(* IEC 61131-3 sources: controlforge-structured-text/manual-tests/diagnostics, 6 files *)

(* ---- array-bounds.st ---- *)
(* Manual QA: array bounds checking for constant indices *)
(* Open this file in VS Code. Verify red squiggles appear ONLY on lines marked  *)
(* "EXPECT ERROR" and that no errors appear on lines marked "OK".               *)
(* Check the Problems panel (Ctrl+Shift+M) for full messages.                   *)

PROGRAM ArrayBoundsTest
VAR
    temps    : ARRAY[1..10] OF REAL;     (* bounds: 1 to 10 *)
    buf      : ARRAY[0..7]  OF BYTE;     (* bounds: 0 to 7  *)
    offsets  : ARRAY[-5..5] OF INT;      (* bounds: -5 to 5 *)
    matrix   : ARRAY[1..4, 1..4] OF REAL; (* 2-D: rows 1-4, cols 1-4 *)
    i        : INT;
    x        : REAL;
END_VAR

    (* --- single-dimension, 1-based --- *)

    (* OK: boundary values *)
    temps[1]  := 20.0;
    temps[10] := 99.9;
    temps[5]  := 50.0;

    (* EXPECT ERROR: index 0 below lower bound 1
       Message: Array index 0 is out of bounds [1..10] for 'temps' *)
    temps[0] := 10.0;

    (* EXPECT ERROR: index 11 above upper bound 10
       Message: Array index 11 is out of bounds [1..10] for 'temps' *)
    temps[11] := 10.0;

    (* EXPECT ERROR: index 15 far above upper bound
       Message: Array index 15 is out of bounds [1..10] for 'temps' *)
    temps[15] := 25.0;

    (* OK: variable index — not checked *)
    temps[i] := 0.0;

    (* --- zero-based array --- *)

    (* OK: valid range *)
    buf[0] := 0;
    buf[7] := 255;

    (* EXPECT ERROR: index 8 above upper bound 7
       Message: Array index 8 is out of bounds [0..7] for 'buf' *)
    buf[8] := 128;

    (* --- negative lower bound --- *)

    (* OK: valid range *)
    offsets[-5] := -1;
    offsets[0]  :=  0;
    offsets[5]  :=  1;

    (* EXPECT ERROR: index -6 below lower bound -5
       Message: Array index -6 is out of bounds [-5..5] for 'offsets' *)
    offsets[-6] := 0;

    (* EXPECT ERROR: index 6 above upper bound 5
       Message: Array index 6 is out of bounds [-5..5] for 'offsets' *)
    offsets[6] := 0;

    (* --- multi-dimensional array --- *)

    (* OK: all indices in range *)
    matrix[1, 1] := 0.0;
    matrix[4, 4] := 1.0;
    matrix[2, 3] := 0.5;

    (* EXPECT ERROR: first index 0 out of [1..4]
       Message: Array index 0 is out of bounds [1..4] for 'matrix' *)
    matrix[0, 2] := 1.0;

    (* EXPECT ERROR: second index 5 out of [1..4]
       Message: Array index 5 is out of bounds [1..4] for 'matrix' *)
    matrix[2, 5] := 1.0;

    (* --- reading (RHS) also checked --- *)

    (* OK *)
    x := temps[3];

    (* EXPECT ERROR: index 99 out of [1..10]
       Message: Array index 99 is out of bounds [1..10] for 'temps' *)
    x := temps[99];

END_PROGRAM

(* ---- assignment-confusion.st ---- *)
(* Manual QA: := vs = confusion detection *)
(* Open this file in VS Code. Verify yellow squiggles (warnings) appear ONLY   *)
(* on lines marked "EXPECT WARNING" and that no warnings appear on "OK" lines. *)
(* For each warning, a lightbulb quick-fix should be available (Ctrl+.).        *)

PROGRAM AssignmentConfusion
VAR
    counter : INT := 0;
    x       : INT := 5;
    ok      : BOOL;
    tmr     : TON;
    arr     : ARRAY[0..9] OF INT;
END_VAR

    (* === Case 1: '=' in statement context — should be ':=' === *)

    (* EXPECT WARNING: "Used '=' in statement context; did you mean ':='?" *)
    (* Quick-fix: Replace '=' with ':='                                    *)
    counter = counter + 1;

    (* EXPECT WARNING *)
    x = 42;

    (* EXPECT WARNING: array element *)
    arr[0] = 5;

    (* OK: correct := assignment — no warning *)
    counter := counter + 1;
    x := 42;
    arr[0] := 5;

    (* OK: '=' in IF condition — intentional comparison *)
    IF x = 10 THEN
        x := 0;
    END_IF;

    (* OK: '=' inside parentheses (RHS comparison) *)
    ok := (x = 5);

    (* OK: '<=' and '>=' — not a bare '=' *)
    ok := x <= 10;
    ok := x >= 0;

    (* OK: '<>' — not a bare '=' *)
    ok := x <> 0;

    (* OK: '=' inside FB call paren (depth > 0) *)
    tmr(IN := TRUE, PT := T#1s);
    IF tmr.Q = TRUE THEN
        tmr(IN := FALSE, PT := T#1s);
    END_IF;

    (* === Case 2: ':=' in boolean condition — should be '=' === *)

    (* EXPECT WARNING: "Used ':=' in condition context; did you mean '='?" *)
    (* Quick-fix: Replace ':=' with '='                                    *)
    IF x := 10 THEN
        x := 0;
    END_IF;

    (* EXPECT WARNING: in ELSIF *)
    IF x = 0 THEN
        x := 1;
    ELSIF x := 5 THEN
        x := 0;
    END_IF;

    (* EXPECT WARNING: in WHILE *)
    WHILE x := 0 DO
        x := x + 1;
    END_WHILE;

    (* OK: correct '=' in IF condition — no warning *)
    IF x = 10 THEN
        x := 0;
    END_IF;

    (* OK: ':=' in FOR loop header is correct syntax — no warning *)
    FOR x := 1 TO 10 DO
        counter := counter + 1;
    END_FOR;

    (* OK: ':=' inside parens in IF body (named parameter) — no warning *)
    IF tmr.Q = TRUE THEN
        tmr(IN := FALSE, PT := T#1s);
    END_IF;

END_PROGRAM

(* ---- code-action-fixes.st ---- *)
(* Test: Code actions for semantic diagnostics *)
(* Open this file, then use Ctrl+. on squiggles to verify quick fixes *)

(* === Insert Semicolon === *)
(* Expected: Quick fix to insert ';' *)
PROGRAM SemicolonFixTest
VAR
    x : INT;
END_VAR
    x := 1  (* <-- hover, Ctrl+. should offer "Insert semicolon" *)
END_PROGRAM

(* === Remove Duplicate Declaration === *)
(* Expected: Quick fix to remove the duplicate line *)
PROGRAM DuplicateFixTest
VAR
    value : INT;
    value : REAL;  (* <-- Ctrl+. should offer "Remove duplicate declaration" *)
END_VAR
    value := 0;
END_PROGRAM

(* === Remove Unused Variable === *)
(* Expected: Quick fix to remove the unused variable line *)
PROGRAM UnusedFixTest
VAR
    active : BOOL;
    unused : INT;  (* <-- Ctrl+. should offer "Remove unused variable" *)
END_VAR
    active := TRUE;
END_PROGRAM

(* ---- constant-assignment.st ---- *)
(* Manual QA: constant assignment detection *)
(* Open this file in VS Code. Verify red squiggles appear ONLY on the lines   *)
(* marked "EXPECT ERROR" and that no errors appear on lines marked "OK".       *)

(* === VAR_GLOBAL CONSTANT === *)
VAR_GLOBAL CONSTANT
    MAX_TEMP : REAL := 100.0;   (* constant — never writable *)
    VERSION  : STRING := 'v1.0';
END_VAR

VAR_GLOBAL
    currentTemp : REAL := 20.0; (* NOT constant — writable *)
END_VAR

(* === PROGRAM body === *)
(* Open this file, then look at the Problems panel (Ctrl+Shift+M).             *)
PROGRAM ConstantTest
VAR CONSTANT
    PI : REAL := 3.14159;       (* local constant *)
END_VAR
VAR
    result : REAL;
    flag   : BOOL;
END_VAR

    (* EXPECT ERROR: Cannot assign to constant 'MAX_TEMP' *)
    MAX_TEMP := 200.0;

    (* EXPECT ERROR: Cannot assign to constant 'PI' *)
    PI := 3.0;

    (* EXPECT ERROR: Cannot assign to constant 'VERSION' *)
    VERSION := 'v2.0';

    (* OK: regular variable assignment — no error *)
    currentTemp := 50.0;
    result := PI * 2.0;         (* reading PI is fine *)
    flag := currentTemp > MAX_TEMP; (* reading constants is fine *)

    (* OK: named FB parameter that happens to use := inside parens — no error *)
    (* (no FB instance here, but illustrates the paren-depth guard)            *)

END_PROGRAM

(* === Verify no false positives for plain VAR_GLOBAL === *)
PROGRAM NoFalsePositives
VAR
    x : REAL;
END_VAR
    (* OK: currentTemp is NOT constant *)
    currentTemp := 99.0;
    x := currentTemp;
END_PROGRAM

(* ---- for-loop-bounds.st ---- *)
(* Manual QA: FOR loop bounds validation *)
(* Open this file in VS Code. Verify squiggles appear ONLY on lines marked     *)
(* "EXPECT <SEVERITY>" and that no squiggles appear on lines marked "OK".      *)
(* Check the Problems panel (Ctrl+Shift+M) for full messages.                   *)

PROGRAM ForLoopBoundsTest
VAR
    i     : INT;
    start : INT;
    stop  : INT;
    total : INT;
END_VAR

    (* ── Normal ascending loops — no diagnostic expected ─────────────────── *)

    (* OK: ascending, default BY (+1) *)
    FOR i := 1 TO 10 DO
        total := total + i;
    END_FOR;

    (* OK: ascending, explicit BY 1 *)
    FOR i := 1 TO 10 BY 1 DO
        total := total + i;
    END_FOR;

    (* OK: descending with BY -1 *)
    FOR i := 10 TO 1 BY -1 DO
        total := total + i;
    END_FOR;

    (* OK: large positive step still valid direction *)
    FOR i := 0 TO 100 BY 5 DO
        total := total + i;
    END_FOR;

    (* OK: variable bounds — not checked at all *)
    FOR i := start TO stop DO
        total := total + i;
    END_FOR;

    (* OK: negative bounds, descending *)
    FOR i := -1 TO -10 BY -1 DO
        total := total + i;
    END_FOR;

    (* ── BY 0: error ─────────────────────────────────────────────────────── *)

    (* EXPECT ERROR on "BY 0": infinite loop
       Problems panel: "FOR loop step BY 0 causes an infinite loop"           *)
    FOR i := 1 TO 10 BY 0 DO
        total := total + i;
    END_FOR;

    (* ── Reverse range with positive BY: warning ─────────────────────────── *)

    (* EXPECT WARNING on "FOR": loop body never executes
       Problems panel: "FOR loop body never executes: counting up (BY 1) but start (10) > end (1)..." *)
    FOR i := 10 TO 1 BY 1 DO
        total := total + i;
    END_FOR;

    (* EXPECT WARNING on "FOR": default BY (+1) with descending range
       Problems panel: "FOR loop body never executes: counting up (BY 1) but start (10) > end (1)..." *)
    FOR i := 10 TO 1 DO
        total := total + i;
    END_FOR;

    (* EXPECT WARNING on "FOR": ascending range with negative step
       Problems panel: "FOR loop body never executes: counting down (BY -2) but start (1) < end (10)..." *)
    FOR i := 1 TO 10 BY -2 DO
        total := total + i;
    END_FOR;

    (* ── Start equals end: hint ──────────────────────────────────────────── *)

    (* EXPECT HINT on "FOR": executes exactly once — likely unintended
       Problems panel: "FOR loop executes exactly once (start equals end: 5)" *)
    FOR i := 5 TO 5 DO
        total := total + i;
    END_FOR;

    (* EXPECT HINT on "FOR": same with explicit BY
       Problems panel: "FOR loop executes exactly once (start equals end: 3)" *)
    FOR i := 3 TO 3 BY 1 DO
        total := total + i;
    END_FOR;

END_PROGRAM

(* ---- semantic-checks.st ---- *)
(* Test: Semantic diagnostics - Phase 2 checks *)
(* Open this file in VS Code to verify diagnostics appear correctly *)

(* === Missing Semicolons === *)
(* Expected: Error on line with missing semicolon *)
PROGRAM MissingSemicolonTest
VAR
    x : INT := 0;
    y : INT := 0;
END_VAR
    x := 1;
    y := x + 2  (* <-- missing semicolon, should show error *)
END_PROGRAM

(* === Duplicate Declarations === *)
(* Expected: Error on second declaration of 'counter' *)
PROGRAM DuplicateVarTest
VAR
    counter : INT;
    counter : REAL;  (* <-- duplicate, should show error *)
    status : BOOL;
END_VAR
    counter := 1;
    status := TRUE;
END_PROGRAM

(* === Undefined Variables === *)
(* Expected: Warning on undeclared identifiers *)
PROGRAM UndefinedVarTest
VAR
    x : INT;
END_VAR
    x := undeclaredVar;  (* <-- undefined, should show warning *)
END_PROGRAM

(* === Unused Variables === *)
(* Expected: Warning on unused local variables *)
PROGRAM UnusedVarTest
VAR
    used : INT;
    unused : INT;  (* <-- never referenced in body, should show warning *)
END_VAR
    used := 42;
END_PROGRAM

(* === Type Mismatches === *)
(* Expected: Error on incompatible assignment *)
PROGRAM TypeMismatchTest
VAR
    count : INT;
    flag : BOOL;
END_VAR
    count := 'hello';  (* <-- STRING to INT, should show error *)
    flag := 42;         (* <-- INT to BOOL, should show error *)
    count := 100;       (* <-- OK, INT to INT *)
    flag := TRUE;       (* <-- OK, BOOL to BOOL *)
END_PROGRAM

(* === Valid Code - No Diagnostics Expected === *)
PROGRAM CleanProgram
VAR
    i : INT;
    sum : INT := 0;
    running : BOOL := TRUE;
END_VAR
    FOR i := 1 TO 10 DO
        sum := sum + i;
    END_FOR
    IF sum > 50 THEN
        running := FALSE;
    END_IF
END_PROGRAM
